SUBAPPLICATION Uebung_020g (* DigitalInput_I1 auf DigitalOutput_Q1; E_TONOF; Ein-/Ausschaltverzögert *)
  (* Standard: 61499-2 *)
  (* Version 1.0, 2023-10-23, franz *)
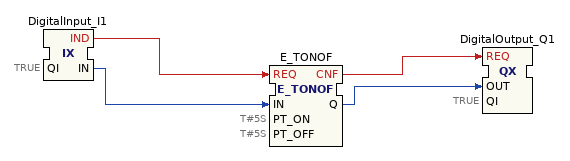
  FBS
    DigitalOutput_Q1 : QX(QI := TRUE);
    DigitalInput_I1 : IX(QI := TRUE);
    E_TONOF : E_TONOF(PT_ON := T#5S, PT_OFF := T#5S);
  END_FBS
  EVENT_CONNECTIONS
    DigitalInput_I1.IND TO E_TONOF.REQ;
    E_TONOF.CNF TO DigitalOutput_Q1.REQ;
  END_CONNECTIONS
  DATA_CONNECTIONS
    DigitalInput_I1.IN TO E_TONOF.IN;
    E_TONOF.Q TO DigitalOutput_Q1.OUT;
  END_CONNECTIONS
END_SUBAPPLICATION
